PROGRAM Firebird_WriteAlarms
VAR_INPUT
	ParamTimeBetweenReconnect	: TIME := T#1M;
	IN_Reset					: BOOL;
	
	FIFO						: FB_DBDatasetFifo;
END_VAR
VAR_OUTPUT
END_VAR
	
VAR

	CmdStart					: BOOL;
	CmdReset					: BOOL;
	// Data processing 
	MesDataExd			: LoggerFirebird ; 
	// RESET
		Trig_Reset				: R_TRIG;
		
	// Connexion
		TP_Reconnect			: TP;
		Trig_Connect			: R_TRIG;
		RS_Connect				: RS;
		RS_HasBeenConnected		: RS;
	// DISCONNECT
		TrigStartDisconnect				: R_TRIG;
		RsStartDisconnect				: RS;		
		
		
	// Write File       
		ETAPE					: UINT;
		Trig_Start				: R_TRIG;   
		Requete					: STRING(1000);
		sTimeStamp 				: STRING(255);
		sTimeStamp_Ms			: STRING(255);
		sValue					: STRING(255);
		sAck					: STRING(255);
		Format					: FB_FormatString;
		SQLDatabase				: FB_SQLDatabaseEvt('',T#10S);
		SQLCommand1				: FB_SQLCommandEvt('',T#10S);
		SQLCommandNull			: FB_SQLCommandEvt('',T#10S);
		
	
	// General variables
		bInit 					: BOOL;

		NomTable				: STRING(255) := 'TABLE_ALARMS';
		

	
END_VAR

// DataProcessing
IF NOT bInit THEN
	M_Init();
END_IF
RS_HasBeenConnected(SET := SQLDatabase.bConnected);
TP_Reconnect(In :=RS_HasBeenConnected.Q1 AND NOT SQLDatabase.bConnected OR NOT bInit OR TP_Reconnect.Q, PT := ParamTimeBetweenReconnect);
	
M_AlarmManager();


Trig_Reset(CLK := IN_Reset OR CmdClearFault_G);
IF Trig_Reset.Q THEN
	FIFO.A_Reset();
	SQLCommand1 := SQLCommandNull;
	CmdReset := False;
END_IF


// La première ligne est non nulle
CmdStart := FIFO.nCount >0 AND SQLDatabase.bConnected;
Trig_Start(CLK := CmdStart);
IF Trig_Start.Q THEN
	ETAPE := 1;
END_IF
		
CASE ETAPE OF
	1: // CONNECTED
		IF SQLDatabase.CreateCmd(pSQLCommand := ADR(SQLCommand1)) THEN 
			IF NOT SQLCommand1.bError THEN
				ETAPE := 2;
			ELSIF SQLCommand1.bError THEN
				ETAPE := 255;
			END_IF
		END_IF
		
	2:
		//sTimeStamp := left(STR := (AX_Buffer_Alarms[1].TimeStamp_Act), SIZE := LEN((AX_Buffer_Alarms[1].TimeStamp_Act))-4);
		FIFO.A_Get();	
		sTimeStamp := FIFO.OUT.TimeStamp_Act;
		sTimeStamp_MS := right(STR := (sTimeStamp), SIZE := 3);	
		sValue	:= INT_TO_STRING(BOOL_TO_INT(FIFO.Out.Value));
		sAck	:= INT_TO_STRING(BOOL_TO_INT(FIFO.Out.Ack));
		Format(sFormat := 'Insert into %s values ( $'%s$',%d, %s, %s);', 
			sOut => Requete,
			arg1 := F_STRING(in := NomTable),
			arg2 := F_STRING(in := sTimeStamp),
			arg3 := F_UINT(in := FIFO.Out.ID),
			arg4 := F_STRING(in := sValue),
			arg5 := F_STRING(in := sAck)
		);
		IF SQLCommand1.Execute(pSQLCmd := ADR(Requete), cbSQLCmd := SIZEOF(Requete))THEN
			IF  NOT SQLCommand1.bError THEN
				ETAPE := 4;
			ELSIF SQLCommand1.bError THEN
				ETAPE := 255;
			END_IF
		END_IF

	4:
		IF NOT SQLDatabase.bError THEN
			FIFO.A_Remove();
			Requete  := '';
			Trig_Start(CLK := FALSE);
			Etape := 0;
		ELSE 
			ETAPE := 255;
		END_IF
		
	255: 
		CmdReset := TRUE;
		Requete := '';
		Etape := 0;
		CmdStart := FALSE;
END_CASE

METHOD M_AlarmManager
VAR
	FB_AlarmCodeManager : FB_AlarmCodeManager;
END_VAR
// Gestion des alarmes internes au code

FB_AlarmCodeManager
(
	bAlarm1 := SQLCommand1.bError,				// Insert new alarm failed
	bAlarm2 := SQLDatabase.bError,				// Connexion to database failed
	bAlarm3 := FALSE,							// 
	bAlarm4 := FIFO.bOverwrite,					// Fifo Overflow
	bAlarm5 :=FALSE,							//
	bAlarm6 :=FALSE,    						//
	bAlarm7 :=FALSE,    						//
	bAlarm8 :=FALSE,    						//
	bAlarm9 :=FALSE,    						//
	bAlarm10 :=FALSE,   						//
	bAlarm11 :=FALSE,   						//
	bAlarm12 :=FALSE,   						//
	bAlarm13 :=FALSE,   						//
	bAlarm14 :=FALSE,   						//
	bAlarm15 :=FALSE,							//	
	
	wAlarmCode =>MesDataExd.MesData.MesAlarmCode
);
END_METHOD

METHOD M_Connect : BOOL

VAR_OUTPUT
END_VAR
VAR_INPUT
	IN_hDBID				: DINT;
	IN_Start				: BOOL;
END_VAR
Trig_Connect(CLK := IN_Start);
RS_Connect(SET := Trig_Connect.Q);
IF RS_Connect.Q1 THEN
	IF SQLDatabase.Connect(hDBID := IN_hDBID) THEN;
		RS_Connect(RESET1 := TRUE);
		RS_Connect(RESET1 := FALSE);
	END_IF
END_IF
END_METHOD

METHOD M_Disconnect : BOOL
VAR_INPUT
END_VAR
VAR_INPUT
	IN_Start				: BOOL;
END_VAR
VAR
END_VAR
TrigStartDisconnect(CLK := IN_Start);
RsStartDisconnect(SET := TrigStartDisconnect.Q);
IF RsStartDisconnect.Q1 THEN
	IF SQLDatabase.Disconnect() THEN;
		RsStartDisconnect(RESET1 := TRUE);
		RsStartDisconnect(RESET1 := FALSE);
	END_IF
END_IF
END_METHOD

METHOD M_Init

VAR
	LL	: SINT;
	KK 	: SINT;
END_VAR
//Initialisation BUFFER
	//Buffer pour la lecture des sms
	FIFO.A_Reset();
	FIFO.A_Add();
	FIFO.A_Get();
	FIFO.A_Remove();
	
	FIFO.In.Message :=  'Activation du code';
	FIFO.In.TimeStamp_Act := SYSTEMTIME_TO_STRING(CalLocalTimeStruct); 
	FIFO.A_Add();
	bInit := TRUE;
END_METHOD

END_PROGRAM

(* stored: Version 1.1.0.1, ProductVersion 3.1.4024.6
   POU Firebird_WriteAlarms: Id {68fbb2cd-160a-435f-85d3-cd562893ee02}, SpecialFunc None
   Method M_AlarmManager: Id {7efc0b73-007b-4998-ba63-127a15bbf9fa}
   Method M_Connect: Id {a3855e20-0182-4f7c-84f5-3d6be1e47f75}
   Method M_Disconnect: Id {dff8ebec-9264-4595-96d7-efee9559e54b}
   Method M_Init: Id {68d5141c-97f6-4519-b39d-92136124bbad} *)
